ABB RobotStudio station: Despending(class 1(robot_15200id)) @ 7020_4.rsstn

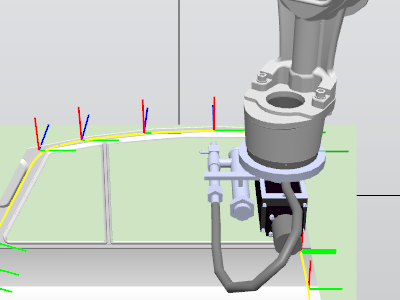
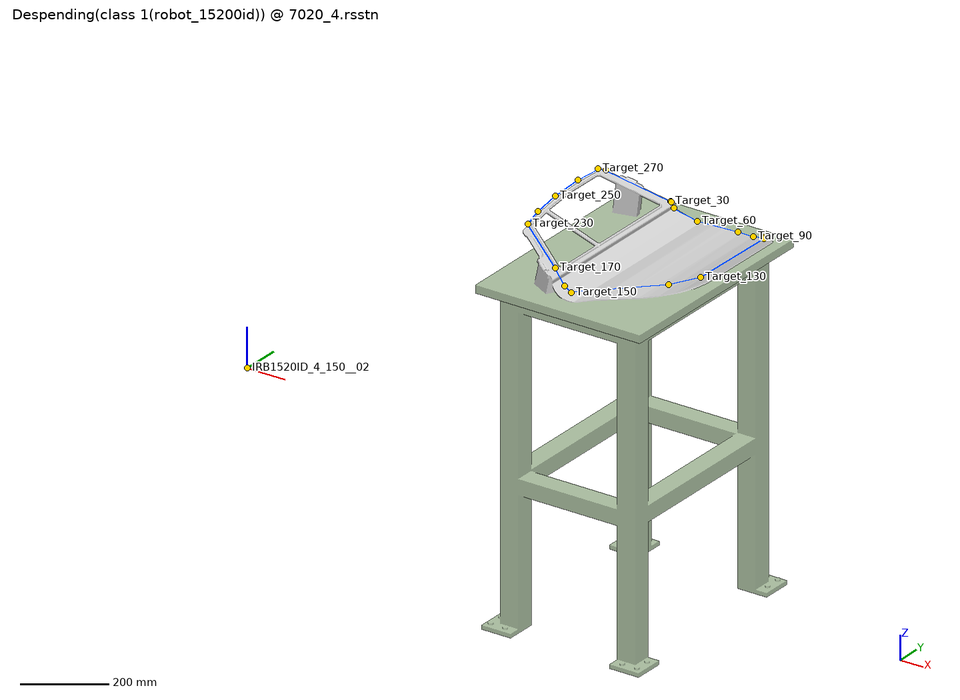
[picture v1: parts stored in the station drawn from their meshes, with robot base, taught points and paths (robot models come from the ABB library and are not in the file)]
Station Despending(class 1(robot_15200id)) @ 7020_3 (saved by RobotStudio 22.3.10141.1)
Controller Controller19, task T_ROB1: task frame (RAPID world) sits at (0, 0, 290) mm in the station
Controller Controller19
  mechanical unit ROB_1: IRB1520ID_4_150__02, 6 joints, base frame (0, 0, 0) mm
Layout (positions relative to the parent item):
  - IRB1520ID_4_150__02 [mechanism, from Robots\IRB1520ID_4_150_G_02.rslib] at (0, 0, 290) mm; joint values [0.2052, -0.3127, 0.6941, -0.8714, 0.2327, 0.9616] (rad or m)
  - Part_1 [part, from Robotics 7020\Cement Base.rslib] at (-450, -450, 0) mm
  - Dispencer [mechanism, from Dispencing\Dispencer.rslib] at (882.01, 147.55, 1120.89) mm, rotated rx -180 ry 60 rz -180 deg
  - table with door [part] at (1436.58, 247.66, 380.24) mm, rotated rx 90 ry 0 rz -90 deg, size 600 x 960.7 x 450 mm
Attachment: Dispencer is attached to IRB1520ID_4_150__02 / Link6
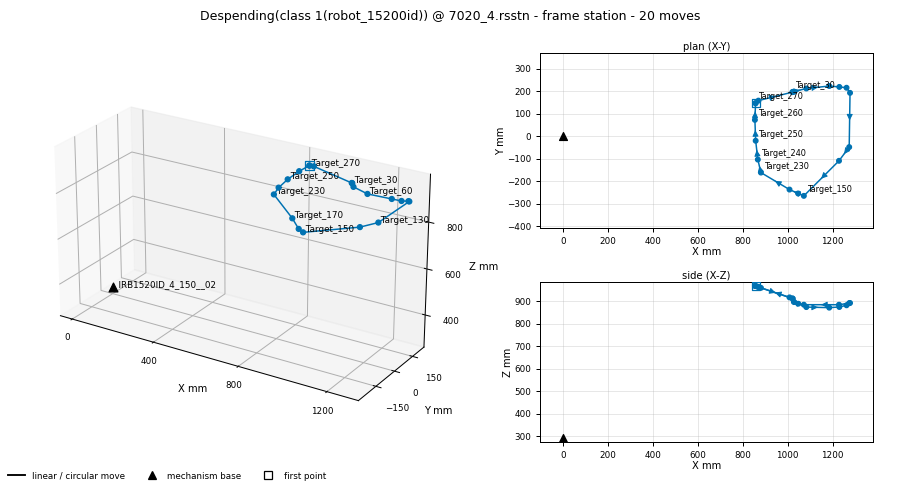
[picture p0: tool path of Despending(class 1(robot_15200id)) @ 7020_4.rsstn in frame station, 20 of 20 moves have a stored position in this frame; points joined in program order, loops and branches not executed]
Targets, tools, work objects and paths stored in the station, written as RAPID:
! task T_ROB1
MODULE CalibData
  PERS tooldata Dispencer:=[TRUE,[[145,-0.097,55],[0.707106781,0,0.707106781,0]],[1,[0,0,1],[1,0,0,0],0,0,0]];
ENDMODULE

! task T_ROB1
MODULE Module1
  CONST robtarget Target_20:=[[870.025900344,159.206036321,673.476082131],[0.258819017,0.000000232,-0.965925834,0.000001089],[0,-1,0,0],[9E+09,9E+09,9E+09,9E+09,9E+09,9E+09]];
  CONST robtarget Target_30:=[[1020.831964931,196.829033591,622.6402853],[0.258819027,0.000000237,-0.965925831,0.000001108],[0,-1,0,0],[9E+09,9E+09,9E+09,9E+09,9E+09,9E+09]];
  CONST robtarget Target_40:=[[1022.855073766,197.333920286,621.958186205],[0.258819021,0.00000024,-0.965925833,0.000001127],[0,-1,0,0],[9E+09,9E+09,9E+09,9E+09,9E+09,9E+09]];
  CONST robtarget Target_50:=[[1027.628174075,199.156727965,606.82760097],[0.2164396,0.000000272,-0.97629601,0.000001083],[0,-2,1,0],[9E+09,9E+09,9E+09,9E+09,9E+09,9E+09]];
  CONST robtarget Target_60:=[[1083.047147401,213.189631292,584.150894588],[0.216439595,0.000000276,-0.976296011,0.000001094],[0,-2,1,0],[9E+09,9E+09,9E+09,9E+09,9E+09,9E+09]];
  CONST robtarget Target_70:=[[1185.066175307,224.077422802,581.628685585],[0.130526174,0.000000367,-0.991444864,0.000001055],[0,-2,1,0],[9E+09,9E+09,9E+09,9E+09,9E+09,9E+09]];
  CONST robtarget Target_90:=[[1230.004260159,220.067029844,584.577400534],[0.130526166,0.000000353,-0.991444865,0.000001035],[0,-2,1,0],[9E+09,9E+09,9E+09,9E+09,9E+09,9E+09]];
  CONST robtarget Target_110:=[[1262.064727943,216.451402766,592.099869547],[0.130526173,0.000000357,-0.991444864,0.000001052],[0,-2,1,0],[9E+09,9E+09,9E+09,9E+09,9E+09,9E+09]];
  CONST robtarget Target_120:=[[1277.63592339,193.677733512,602.424532716],[0.130526179,0.000000343,-0.991444863,0.000001015],[0,-2,1,0],[9E+09,9E+09,9E+09,9E+09,9E+09,9E+09]];
  CONST robtarget Target_140:=[[1228.50030933,-108.760570161,594.664916557],[0.128543018,-0.172162274,-0.976382645,0.02266658],[-1,-2,1,0],[9E+09,9E+09,9E+09,9E+09,9E+09,9E+09]];
  CONST robtarget Target_150:=[[1072.097028239,-264.712215107,594.75633135],[0.2548868,-0.167731072,-0.951251284,0.044944426],[-1,-2,1,0],[9E+09,9E+09,9E+09,9E+09,9E+09,9E+09]];
  CONST robtarget Target_160:=[[1046.729697332,-254.042714244,599.052691876],[0.254886798,-0.167731054,-0.951251287,0.044944443],[-1,-2,1,0],[9E+09,9E+09,9E+09,9E+09,9E+09,9E+09]];
  CONST robtarget Target_230:=[[881.070798953,-161.173257724,669.75285346],[0.258819026,0.000000187,-0.965925831,0.000000901],[-1,0,-1,0],[9E+09,9E+09,9E+09,9E+09,9E+09,9E+09]];
  CONST robtarget Target_240:=[[867.280312505,-103.210959469,674.401599165],[0.258819027,0.000000182,-0.965925831,0.000000871],[-1,0,-1,0],[9E+09,9E+09,9E+09,9E+09,9E+09,9E+09]];
  CONST robtarget Target_250:=[[857.67074272,-19.504931503,677.641008777],[0.258819021,0.000000182,-0.965925833,0.000000872],[-1,0,-1,0],[9E+09,9E+09,9E+09,9E+09,9E+09,9E+09]];
  CONST robtarget Target_260:=[[854.194884655,73.514086147,678.812688959],[0.258819033,0.000000191,-0.965925829,0.000000914],[0,-1,0,0],[9E+09,9E+09,9E+09,9E+09,9E+09,9E+09]];
  CONST robtarget Target_270:=[[857.138298979,147.455518064,677.820481401],[0.258819023,0.000000187,-0.965925832,0.000000911],[0,-1,0,0],[9E+09,9E+09,9E+09,9E+09,9E+09,9E+09]];
  CONST robtarget Target_130:=[[1273.922734782,-47.688873144,601.474970182],[0.129525198,-0.122556399,-0.983840866,-0.016133923],[0,-2,1,0],[9E+09,9E+09,9E+09,9E+09,9E+09,9E+09]];
  CONST robtarget Target_170:=[[1008.251036482,-236.70553257,627.237004474],[0.254886795,-0.167731006,-0.951251295,0.044944459],[-1,-1,0,0],[9E+09,9E+09,9E+09,9E+09,9E+09,9E+09]];
  PROC Path_10()
    MoveL Target_270,v1000,z100,Dispencer\WObj:=wobj0;
    MoveL Target_20,v1000,z100,Dispencer\WObj:=wobj0;
    MoveL Target_30,v1000,z100,Dispencer\WObj:=wobj0;
    MoveL Target_40,v1000,z100,Dispencer\WObj:=wobj0;
    MoveL Target_50,v1000,z100,Dispencer\WObj:=wobj0;
    MoveL Target_60,v1000,z100,Dispencer\WObj:=wobj0;
    MoveL Target_70,v1000,z100,Dispencer\WObj:=wobj0;
    MoveL Target_90,v1000,z100,Dispencer\WObj:=wobj0;
    MoveL Target_110,v1000,z100,Dispencer\WObj:=wobj0;
    MoveL Target_120,v1000,z100,Dispencer\WObj:=wobj0;
    MoveL Target_130,v1000,z100,Dispencer\WObj:=wobj0;
    MoveL Target_140,v1000,z100,Dispencer\WObj:=wobj0;
    MoveL Target_150,v1000,z100,Dispencer\WObj:=wobj0;
    MoveL Target_160,v1000,z100,Dispencer\WObj:=wobj0;
    MoveL Target_170,v1000,z100,Dispencer\WObj:=wobj0;
    MoveL Target_230,v1000,z100,Dispencer\WObj:=wobj0;
    MoveL Target_240,v1000,z100,Dispencer\WObj:=wobj0;
    MoveL Target_250,v1000,z100,Dispencer\WObj:=wobj0;
    MoveL Target_260,v1000,z100,Dispencer\WObj:=wobj0;
    MoveL Target_270,v1000,z100,Dispencer\WObj:=wobj0;
  ENDPROC
ENDMODULE

